{attribute 'qualified_only'}
{attribute 'strict'}
TYPE TaitBryanAngleSequence :
(
	XYZ := 0,
	YZX := 1,
	ZXY := 2,
	XZY := 3,
	ZYX := 4,
	YXZ := 5	//Standard Roll/Pitch/Yaw
);
END_TYPE

(* stored: Version 1.1.0.1, ProductVersion 3.1.4024.9
   DUT TaitBryanAngleSequence: Id {77e645ed-c33e-0fe4-130a-e049a56d9045} *)
